// TIA Portal V18 export
FUNCTION "HVACGeneralParams" : Void   // FC99, LAD
{ S7_Optimized_Access := 'TRUE' }
VERSION : 0.1
// stored: AutoNumber false, IsIECCheckEnabled false, SetENOAutomatically false, UDAEnableTagReadback false
BEGIN

REGION Network 1 (SCL): Season Target
   CASE "HVAC_Vars".Season.cSeasonModeSelection OF
       0:  // Summer;
           "HVAC_Vars".Season.cTarget := 0;
       1:  // Winter
           "HVAC_Vars".Season.cTarget := 1;
       2:  // Midseason
           "HVAC_Vars".Season.cTarget := 2;
       ELSE  // Auto by OAT
           IF "OAT".Temp.rOAT_Actual < "HVAC_Vars".Season.rOATtoWinter THEN
               "HVAC_Vars".Season.cTarget := 1;
           ELSIF "OAT".Temp.rOAT_Actual > "HVAC_Vars".Season.rOATtoSummer THEN
               "HVAC_Vars".Season.cTarget := 0;
           END_IF;
   END_CASE;
END_REGION

REGION Network 2 (SCL): Season Actual
   "HVAC_Vars".Season.cActual := "HVAC_Vars".Season.cTarget;
END_REGION

REGION Network 3: Розклад
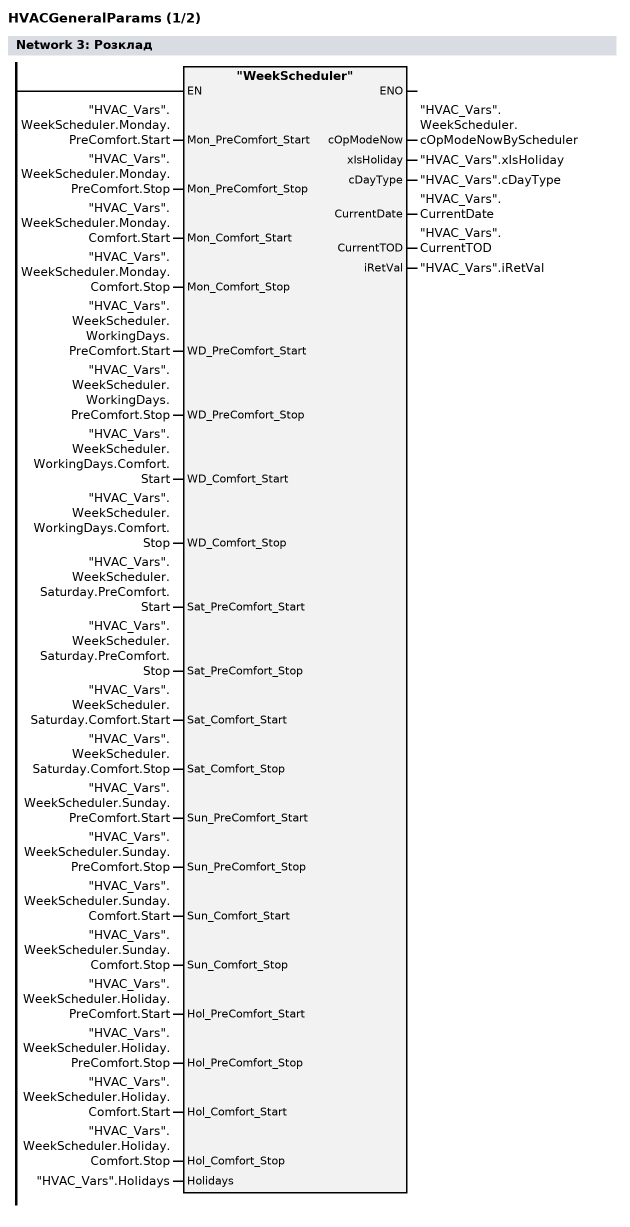
   RUNG wire#powerrail
      "WeekScheduler"(Mon_PreComfort_Start := "HVAC_Vars".WeekScheduler.Monday.PreComfort.Start, Mon_PreComfort_Stop := "HVAC_Vars".WeekScheduler.Monday.PreComfort.Stop, Mon_Comfort_Start := "HVAC_Vars".WeekScheduler.Monday.Comfort.Start, Mon_Comfort_Stop := "HVAC_Vars".WeekScheduler.Monday.Comfort.Stop, WD_PreComfort_Start := "HVAC_Vars".WeekScheduler.WorkingDays.PreComfort.Start, WD_PreComfort_Stop := "HVAC_Vars".WeekScheduler.WorkingDays.PreComfort.Stop, WD_Comfort_Start := "HVAC_Vars".WeekScheduler.WorkingDays.Comfort.Start, WD_Comfort_Stop := "HVAC_Vars".WeekScheduler.WorkingDays.Comfort.Stop, Sat_PreComfort_Start := "HVAC_Vars".WeekScheduler.Saturday.PreComfort.Start, Sat_PreComfort_Stop := "HVAC_Vars".WeekScheduler.Saturday.PreComfort.Stop, Sat_Comfort_Start := "HVAC_Vars".WeekScheduler.Saturday.Comfort.Start, Sat_Comfort_Stop := "HVAC_Vars".WeekScheduler.Saturday.Comfort.Stop, Sun_PreComfort_Start := "HVAC_Vars".WeekScheduler.Sunday.PreComfort.Start, Sun_PreComfort_Stop := "HVAC_Vars".WeekScheduler.Sunday.PreComfort.Stop, Sun_Comfort_Start := "HVAC_Vars".WeekScheduler.Sunday.Comfort.Start, Sun_Comfort_Stop := "HVAC_Vars".WeekScheduler.Sunday.Comfort.Stop, Hol_PreComfort_Start := "HVAC_Vars".WeekScheduler.Holiday.PreComfort.Start, Hol_PreComfort_Stop := "HVAC_Vars".WeekScheduler.Holiday.PreComfort.Stop, Hol_Comfort_Start := "HVAC_Vars".WeekScheduler.Holiday.Comfort.Start, Hol_Comfort_Stop := "HVAC_Vars".WeekScheduler.Holiday.Comfort.Stop, Holidays := "HVAC_Vars".Holidays, cOpModeNow => "HVAC_Vars".WeekScheduler.cOpModeNowByScheduler, xIsHoliday => "HVAC_Vars".xIsHoliday, cDayType => "HVAC_Vars".cDayType, CurrentDate => "HVAC_Vars".CurrentDate, CurrentTOD => "HVAC_Vars".CurrentTOD, iRetVal => "HVAC_Vars".iRetVal)
   END_RUNG
   // the same network as SCL:
   "WeekScheduler"(Mon_PreComfort_Start := "HVAC_Vars".WeekScheduler.Monday.PreComfort.Start,
                   Mon_PreComfort_Stop := "HVAC_Vars".WeekScheduler.Monday.PreComfort.Stop,
                   Mon_Comfort_Start := "HVAC_Vars".WeekScheduler.Monday.Comfort.Start,
                   Mon_Comfort_Stop := "HVAC_Vars".WeekScheduler.Monday.Comfort.Stop,
                   WD_PreComfort_Start := "HVAC_Vars".WeekScheduler.WorkingDays.PreComfort.Start,
                   WD_PreComfort_Stop := "HVAC_Vars".WeekScheduler.WorkingDays.PreComfort.Stop,
                   WD_Comfort_Start := "HVAC_Vars".WeekScheduler.WorkingDays.Comfort.Start,
                   WD_Comfort_Stop := "HVAC_Vars".WeekScheduler.WorkingDays.Comfort.Stop,
                   Sat_PreComfort_Start := "HVAC_Vars".WeekScheduler.Saturday.PreComfort.Start,
                   Sat_PreComfort_Stop := "HVAC_Vars".WeekScheduler.Saturday.PreComfort.Stop,
                   Sat_Comfort_Start := "HVAC_Vars".WeekScheduler.Saturday.Comfort.Start,
                   Sat_Comfort_Stop := "HVAC_Vars".WeekScheduler.Saturday.Comfort.Stop,
                   Sun_PreComfort_Start := "HVAC_Vars".WeekScheduler.Sunday.PreComfort.Start,
                   Sun_PreComfort_Stop := "HVAC_Vars".WeekScheduler.Sunday.PreComfort.Stop,
                   Sun_Comfort_Start := "HVAC_Vars".WeekScheduler.Sunday.Comfort.Start,
                   Sun_Comfort_Stop := "HVAC_Vars".WeekScheduler.Sunday.Comfort.Stop,
                   Hol_PreComfort_Start := "HVAC_Vars".WeekScheduler.Holiday.PreComfort.Start,
                   Hol_PreComfort_Stop := "HVAC_Vars".WeekScheduler.Holiday.PreComfort.Stop,
                   Hol_Comfort_Start := "HVAC_Vars".WeekScheduler.Holiday.Comfort.Start,
                   Hol_Comfort_Stop := "HVAC_Vars".WeekScheduler.Holiday.Comfort.Stop,
                   Holidays := "HVAC_Vars".Holidays,
                   cOpModeNow => "HVAC_Vars".WeekScheduler.cOpModeNowByScheduler,
                   xIsHoliday => "HVAC_Vars".xIsHoliday,
                   cDayType => "HVAC_Vars".cDayType,
                   CurrentDate => "HVAC_Vars".CurrentDate,
                   CurrentTOD => "HVAC_Vars".CurrentTOD,
                   iRetVal => "HVAC_Vars".iRetVal);
END_REGION

REGION Network 4 (SCL): OpMode Target
   CASE "HVAC_Vars".OpModes.cPreselectedOpMode OF
       0:  // Protection;
           "HVAC_Vars".OpModes.cTarget := 0;
       1:  // Economy
           "HVAC_Vars".OpModes.cTarget := 1;
       2:  // PreComf
           "HVAC_Vars".OpModes.cTarget := 2;
       3:  // Comf
           "HVAC_Vars".OpModes.cTarget := 3;
       ELSE  // Auto by Scheduler
           "HVAC_Vars".OpModes.cTarget := "HVAC_Vars".WeekScheduler.cOpModeNowByScheduler;
   END_CASE;
END_REGION

REGION Network 5 (SCL): OpMode Actual
   "HVAC_Vars".OpModes.cActual := "HVAC_Vars".OpModes.cTarget;
END_REGION

REGION Network 6 (SCL): Temp Setpoints to schow on HMI
   CASE "HVAC_Vars".Season.cActual OF
       0:  // Summer
           "HVAC_Vars".RoomTempSetPointforHMI := "HVAC_Vars".SetPoints.Room.Actual.rRATCooling;
       1:  // Winter
           "HVAC_Vars".RoomTempSetPointforHMI := "HVAC_Vars".SetPoints.Room.Actual.rRATHeating;
       ELSE  // Statement section ELSE
           "HVAC_Vars".RoomTempSetPointforHMI := ("HVAC_Vars".SetPoints.Room.Actual.rRATHeating+"HVAC_Vars".SetPoints.Room.Actual.rRATCooling)/2;
   END_CASE;
END_REGION

REGION Network 7 (SCL): Actual OAT
   CASE "OAT".cSelectOATMode OF
       0:
           "OAT".Temp.rOAT_Actual := "HSsAI".AI.rOutdoorTemp_PLC_AI;
       1:
           "OAT".Temp.rOAT_Actual := "OAT".Temp.rOAT_WeatherStation;
       2:
           "OAT".Temp.rOAT_Actual := "OAT".Temp.rOAT_Boilers;
       ELSE  // Statement section ELSE
           "OAT".Temp.rOAT_Actual := "OAT".Temp.rOAT_PLC_IO;
   END_CASE;
END_REGION

REGION Network 8 (SCL): Select values for Actual SP
   CASE "HVAC_Vars".OpModes.cActual OF
       0:  // Protection mode
           "HVAC_Vars".SetPoints.Room.Actual.rRATHeating := "HVAC_Vars".SetPoints.Room.Protection.rRATHeating;
           "HVAC_Vars".SetPoints.Room.Actual.rRATCooling := "HVAC_Vars".SetPoints.Room.Protection.rRATCooling;
           "HVAC_Vars".SetPoints.Room.Actual.rIAQ := "HVAC_Vars".SetPoints.Room.Protection.rIAQ;
           "HVAC_Vars".SetPoints.Room.Actual.rBuildingdP := "HVAC_Vars".SetPoints.Room.Protection.rBuildingdP;
       1:  // Economy mode
           "HVAC_Vars".SetPoints.Room.Actual.rRATHeating := "HVAC_Vars".SetPoints.Room.Econom.rRATHeating;
           "HVAC_Vars".SetPoints.Room.Actual.rRATCooling := "HVAC_Vars".SetPoints.Room.Econom.rRATCooling;
           "HVAC_Vars".SetPoints.Room.Actual.rIAQ := "HVAC_Vars".SetPoints.Room.Econom.rIAQ;
           "HVAC_Vars".SetPoints.Room.Actual.rBuildingdP := "HVAC_Vars".SetPoints.Room.Econom.rBuildingdP;
       2:  // PreComfort mode
           "HVAC_Vars".SetPoints.Room.Actual.rRATHeating := "HVAC_Vars".SetPoints.Room.PreComfort.rRATHeating;
           "HVAC_Vars".SetPoints.Room.Actual.rRATCooling := "HVAC_Vars".SetPoints.Room.PreComfort.rRATCooling;
           "HVAC_Vars".SetPoints.Room.Actual.rIAQ := "HVAC_Vars".SetPoints.Room.PreComfort.rIAQ;
           "HVAC_Vars".SetPoints.Room.Actual.rBuildingdP := "HVAC_Vars".SetPoints.Room.PreComfort.rBuildingdP;
       3:  // Comfort mode
           "HVAC_Vars".SetPoints.Room.Actual.rRATHeating := "HVAC_Vars".SetPoints.Room.Comfort.rRATHeating;
           "HVAC_Vars".SetPoints.Room.Actual.rRATCooling := "HVAC_Vars".SetPoints.Room.Comfort.rRATCooling;
           "HVAC_Vars".SetPoints.Room.Actual.rIAQ := "HVAC_Vars".SetPoints.Room.Comfort.rIAQ;
           "HVAC_Vars".SetPoints.Room.Actual.rBuildingdP := "HVAC_Vars".SetPoints.Room.Comfort.rBuildingdP;
   END_CASE;
END_REGION

REGION Network 9 (SCL)
   //IF "AHUOpModes".OpModes.cActual[#iUnitID] = "AHUOpModes".OpModes.cTarget[#iUnitID] THEN // !!!Змінити на PrevOpMode
   //    // Statement section IF
   //   CASE "AHUOpModes".OpModes.cActual[#iUnitID] OF
   //        0:  // Protection
   //            "AHUSetPoints".SetPoints.Room.Target.RATHeating[#iUnitID] := #rActualStoreSPTempHeating;
   //            "AHUSetPoints".SetPoints.Room.Target.RATCooling[#iUnitID] := #rActualStoreSPTempCooling;
   //            "AHUSetPoints".SetPoints.Room.Target.IAQ[#iUnitID] := #rActualStoreSPIAQ;
   //            "AHUSetPoints".SetPoints.Room.Target.BuildingdP[#iUnitID] := #rActualStoreSPdP;
   //        1:  // Economy
   //            "AHUSetPoints".SetPoints.Room.Target.RATHeating[#iUnitID] := #rEconTempHeating;
   //            "AHUSetPoints".SetPoints.Room.Target.RATCooling[#iUnitID] := #rEconTempCooling;
   //            "AHUSetPoints".SetPoints.Room.Target.IAQ[#iUnitID] := #rEconIAQ;
   //            "AHUSetPoints".SetPoints.Room.Target.BuildingdP[#iUnitID] := #rAHUShiftTempCoolingSP;
   //        2: // Precomfort
   //            "AHUSetPoints".SetPoints.Room.Target.RATHeating[#iUnitID] := #rPreComfTempHeating;
   //            "AHUSetPoints".SetPoints.Room.Target.RATCooling[#iUnitID] := #rPreComfTempCooling;
   //            "AHUSetPoints".SetPoints.Room.Target.IAQ[#iUnitID] := #rPreComfIAQ;
   //            "AHUSetPoints".SetPoints.Room.Target.BuildingdP[#iUnitID] := #rAHUShiftIAQSP;
   //        ELSE  // Statement section ELSE
   //            "AHUSetPoints".SetPoints.Room.Target.RATHeating[#iUnitID] := #rComfTempHeating;
   //            "AHUSetPoints".SetPoints.Room.Target.RATCooling[#iUnitID] := #rComfTempCooling;
   //            "AHUSetPoints".SetPoints.Room.Target.IAQ[#iUnitID] := #rComfIAQ;
   //            "AHUSetPoints".SetPoints.Room.Target.BuildingdP[#iUnitID] := #rAHUShiftdPSP;
   //    END_CASE;
   //    ;
   //END_IF;
END_REGION

REGION Network 10: Weather Depend Calc. Boiler Setpoint
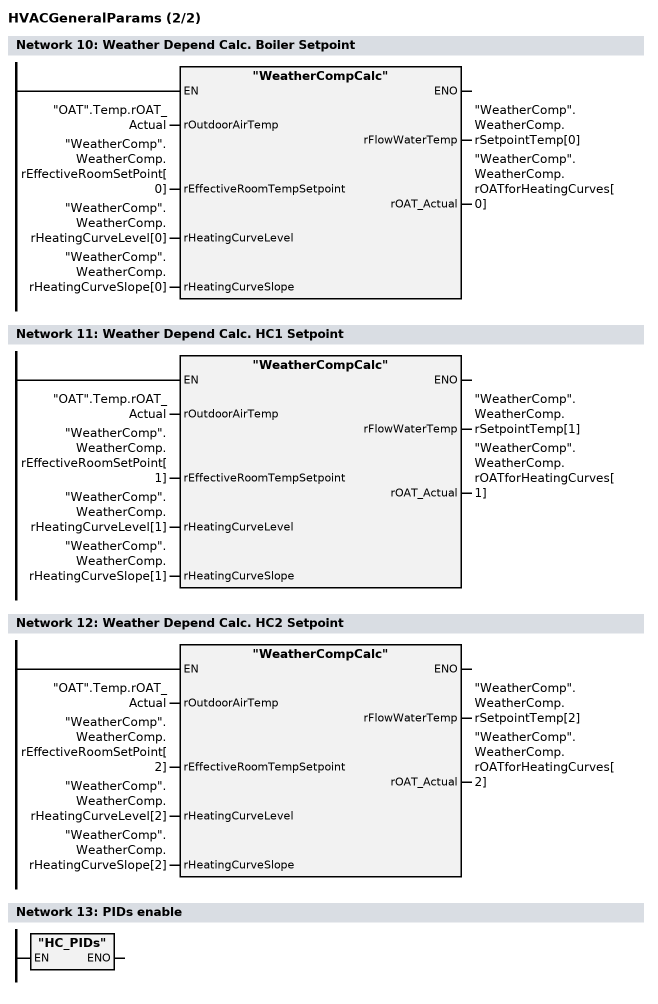
   RUNG wire#powerrail
      "WeatherCompCalc"(rOutdoorAirTemp := "OAT".Temp.rOAT_Actual, rEffectiveRoomTempSetpoint := "WeatherComp".WeatherComp.rEffectiveRoomSetPoint[0], rHeatingCurveLevel := "WeatherComp".WeatherComp.rHeatingCurveLevel[0], rHeatingCurveSlope := "WeatherComp".WeatherComp.rHeatingCurveSlope[0], rFlowWaterTemp => "WeatherComp".WeatherComp.rSetpointTemp[0], rOAT_Actual => "WeatherComp".WeatherComp.rOATforHeatingCurves[0])
   END_RUNG
   // the same network as SCL:
   "WeatherCompCalc"(rOutdoorAirTemp := "OAT".Temp.rOAT_Actual,
                     rEffectiveRoomTempSetpoint := "WeatherComp".WeatherComp.rEffectiveRoomSetPoint[0],
                     rHeatingCurveLevel := "WeatherComp".WeatherComp.rHeatingCurveLevel[0],
                     rHeatingCurveSlope := "WeatherComp".WeatherComp.rHeatingCurveSlope[0],
                     rFlowWaterTemp => "WeatherComp".WeatherComp.rSetpointTemp[0],
                     rOAT_Actual => "WeatherComp".WeatherComp.rOATforHeatingCurves[0]);
END_REGION

REGION Network 11: Weather Depend Calc. HC1 Setpoint
   RUNG wire#powerrail
      "WeatherCompCalc"(rOutdoorAirTemp := "OAT".Temp.rOAT_Actual, rEffectiveRoomTempSetpoint := "WeatherComp".WeatherComp.rEffectiveRoomSetPoint[1], rHeatingCurveLevel := "WeatherComp".WeatherComp.rHeatingCurveLevel[1], rHeatingCurveSlope := "WeatherComp".WeatherComp.rHeatingCurveSlope[1], rFlowWaterTemp => "WeatherComp".WeatherComp.rSetpointTemp[1], rOAT_Actual => "WeatherComp".WeatherComp.rOATforHeatingCurves[1])
   END_RUNG
   // the same network as SCL:
   "WeatherCompCalc"(rOutdoorAirTemp := "OAT".Temp.rOAT_Actual,
                     rEffectiveRoomTempSetpoint := "WeatherComp".WeatherComp.rEffectiveRoomSetPoint[1],
                     rHeatingCurveLevel := "WeatherComp".WeatherComp.rHeatingCurveLevel[1],
                     rHeatingCurveSlope := "WeatherComp".WeatherComp.rHeatingCurveSlope[1],
                     rFlowWaterTemp => "WeatherComp".WeatherComp.rSetpointTemp[1],
                     rOAT_Actual => "WeatherComp".WeatherComp.rOATforHeatingCurves[1]);
END_REGION

REGION Network 12: Weather Depend Calc. HC2 Setpoint
   RUNG wire#powerrail
      "WeatherCompCalc"(rOutdoorAirTemp := "OAT".Temp.rOAT_Actual, rEffectiveRoomTempSetpoint := "WeatherComp".WeatherComp.rEffectiveRoomSetPoint[2], rHeatingCurveLevel := "WeatherComp".WeatherComp.rHeatingCurveLevel[2], rHeatingCurveSlope := "WeatherComp".WeatherComp.rHeatingCurveSlope[2], rFlowWaterTemp => "WeatherComp".WeatherComp.rSetpointTemp[2], rOAT_Actual => "WeatherComp".WeatherComp.rOATforHeatingCurves[2])
   END_RUNG
   // the same network as SCL:
   "WeatherCompCalc"(rOutdoorAirTemp := "OAT".Temp.rOAT_Actual,
                     rEffectiveRoomTempSetpoint := "WeatherComp".WeatherComp.rEffectiveRoomSetPoint[2],
                     rHeatingCurveLevel := "WeatherComp".WeatherComp.rHeatingCurveLevel[2],
                     rHeatingCurveSlope := "WeatherComp".WeatherComp.rHeatingCurveSlope[2],
                     rFlowWaterTemp => "WeatherComp".WeatherComp.rSetpointTemp[2],
                     rOAT_Actual => "WeatherComp".WeatherComp.rOATforHeatingCurves[2]);
END_REGION

REGION Network 13: PIDs enable
   RUNG wire#powerrail
      "HC_PIDs"()
   END_RUNG
   // the same network as SCL:
   "HC_PIDs"();
END_REGION
END_FUNCTION
